Staubli VAL3: resetnum.pgx

program resetnum(num x_nNum1 (dimensions=1))
begin
  //  //  while size(pCreatTest)>x_nNum1
  //  //    $ddel(pCreatTest,size(pCreatTest)-1)
  //  //  endWhile
  //  //  while size(pCreatTest)<x_nNum1
  //  //    $dins(pCreatTest,size(pCreatTest))
  //  //  endWhile
  //  if x_nNum1>0
  //    while size(cad:pCad)>x_nNum1
  //      $ddel(cad:pCad,size(cad:pCad)-1)
  //      //$ddel(jJointRx,size(jJointRx)-1)
  //    endWhile
  //    while size(cad:jJointRx)>x_nNum1
  //      //$ddel(cad:pCad,size(cad:pCad)-1)
  //      $ddel(cad:jJointRx,size(cad:jJointRx)-1)
  //    endWhile
  //    while size(cad:jJointRx)<x_nNum1
  //      //$dins(cad:pCad,size(cad:pCad))
  //      $dins(cad:jJointRx,size(cad:jJointRx))
  //    endWhile
  //    while size(cad:pCad)<x_nNum1
  //      $dins(cad:pCad,size(cad:pCad))
  //      //$dins(jJointRx,size(jJointRx))
  //    endWhile
  //  else
  //    popUpMsg("点数应大于0")
  //  endIf
end
